Staubli VAL3: initParams.pgx

public program initParams()
  local num l_nRetVal
begin
  // Copyright (c) 2016, Ocado Technology - Robotics Research Team
  // Copyright (c) 2021, Institute for Factory Automation and Production Systems (FAPS)
  //
  // Licensed under the Apache License, Version 2.0 (the "License");
  // you may not use this file except in compliance with the License.
  // You may obtain a copy of the License at
  //
  //     http://www.apache.org/licenses/LICENSE-2.0
  //
  // Unless required by applicable law or agreed to in writing, software
  // distributed under the License is distributed on an "AS IS" BASIS,
  // WITHOUT WARRANTIES OR CONDITIONS OF ANY KIND, either express or implied.
  // See the License for the specific language governing permissions and
  // limitations under the License.

  MsgRecvState.RECEIVE_HEADER=0
  MsgRecvState.DECODE_HEADER=1
  MsgRecvState.RECEIVE_BODY=2
  MsgRecvState.DECODE_BODY=3
  MsgRecvState.PUSH_MOTION=4
  MsgRecvState.HANDLE_REQUEST=5
  MsgRecvState.SEND_ACK=6

  l_nRetVal=sioCtrl(siTcpIpIO,"timeout",-1)
  if (l_nRetVal!=0)
    popUpMsg("Error while setting 'IO' socket timeout")
  endIf

  l_nRetVal=sioCtrl(siTcpIpMotion,"timeout",-1)
  if (l_nRetVal!=0)
    popUpMsg("Error while setting 'Motion' socket timeout")
  endIf

  l_nRetVal=sioCtrl(siTcpIpState,"timeout",-1)
  if (l_nRetVal!=0)
    popUpMsg("Error while setting 'State' socket timeout")
  endIf

  l_nRetVal=sioCtrl(siTcpIpSystem,"timeout",-1)
  if (l_nRetVal!=0)
    popUpMsg("Error while setting 'System' socket timeout")
  endIf
end
